// TIA Portal V21 export
VAR_GLOBAL   // PLC tag table "GruppoRiempiSendAnalogici"
END_VAR
VAR_GLOBAL CONSTANT   // user constants
   K_SegnaleVersoGruppoRiempi_TemperaturaEsercizio : Int := 1;
END_VAR
